// TIA Portal V19 export
VAR_GLOBAL   // PLC tag table "Default tag table"
   Tag_1 AT %M0.5 : Bool;
   Clock_Byte AT %MB0 : Byte;
   Clock_10Hz AT %M0.0 : Bool;
   Clock_5Hz AT %M0.1 : Bool;
   "Clock_2.5Hz" AT %M0.2 : Bool;
   Clock_2Hz AT %M0.3 : Bool;
   "Clock_1.25Hz" AT %M0.4 : Bool;
   Clock_1Hz AT %M0.5 : Bool;
   "Clock_0.625Hz" AT %M0.6 : Bool;
   "Clock_0.5Hz" AT %M0.7 : Bool;
   VibSensor01 AT %I100.0 : "PII - BCM R15E-001-DI00-01,5-S4";
   VibSensor02 AT %I124.0 : "PII - BCM R15E-001-DI00-01,5-S4";
   VibSensor03 AT %I148.0 : "PII - BCM R15E-001-DI00-01,5-S4";
   TempHumidSensor01 AT %I172.0 : "PII - CSS 01411.2-xx";
   OilContaminationSensor01 AT %I184.0 : "PII - BCI24-DH367-1D1A-4";
   AirFlowSensor01 AT %I194.0 : "PII - AS5-AF2-FLX-G100";
END_VAR
